FUNCTION_BLOCK PalletizerRemoteCtrl
VAR_INPUT
	bExecute : BOOL;
END_VAR
VAR_IN_OUT
	fbPalletizer : Palletizer;
END_VAR
VAR_OUTPUT
END_VAR
VAR
	
	udiStep : UDINT;
	messageIndex : UINT;
	remoteCtrlPayload : ST_MqttPayload;
	
	eActuatorType : E_ActuatorType;

END_VAR

(*

Description:
========================================================================	
	
	+	check if AdsConnector is connected
	+	if connected, subscribe to PalHmi topic
	+	check for incoming messages
	+	if message available, check message type 
	+	possible message types are:
	
			+	mode manual
			
				+	actuator type
				
					+	Belt
						+	forware
						+	backward
						
					+	Chain
						+	forward
						+	backward	
						
					+	BeltConveyor
						+	forward
						+	backward
						+	velocity
						
					+	RollerConveyor
						+	forward
						+	backward
						+	velocity	
						
					+	Turn
						+	forward
						+	backward
						
					+	Clamper
						+	clamp
						+	unclamp
	
					+	Pusher
						+	push forward
						+	push backward
						
					+	Plate
						+	open plate
						+	close plate
						
					+	Elevator
						+	up
						+	down
						+	to limit
						
			+	mode automatic
				
				+	start
				+	stop
			
			+	mode system
			
				+	home
				+	reset
				
			
=========================================================================

*)



IF 	ADS.fbAdsConnector.isConnected
	AND bExecute
THEN

	udiStep := 10;
ELSE
	udiStep := 0;
END_IF

CASE udiStep OF

	10:
		IF ADS.fbMqttClient.subscribe('PalHmi',THIS)
		THEN
			udiStep := 20;
		END_IF
		
	20:
		messageIndex := ADS.fbMqttClient.isNewMessage('PalHmi');
		IF messageIndex > 0
		THEN
		
			evaluateMode(Ads.fbMqttClient.getNewMessage(messageIndex));
			
		END_IF
			
		
END_CASE

METHOD PRIVATE evaluateActuator : BOOL
VAR_INPUT
	remoteCtrlPayload : ST_MqttPayload;
END_VAR
VAR
	eCmd : E_ActuatorCmdType;
	eActuator : E_ActuatorType;
END_VAR
eActuator := BYTE_TO_UINT(remoteCtrlPayload.data[2]);
eCmd := BYTE_TO_UINT(remoteCtrlPayload.data[3]);

CASE eActuator OF

	ePALLETIZER_BELT:
		
		fbPalletizer.fbBeltConveyor.cmd := eCmd;
		
	ePALLETIZER_CHAIN:
	
		fbPalletizer.fbPalletizerChain.cmd := eCmd;
		
	eBELT_CONVEYOR:
		
		fbPalletizer.fbBeltConveyor.cmd := eCmd;
		
	eROLLER_CONVEYOR:
		
		fbPalletizer.fbRollerConveyor.cmd := eCmd;
		
	eTURN_CYLINDER:
		
		fbPalletizer.fbTurnCylinder.cmd := eCmd;
	
	eCLAMPER_CYLINDER:
		
		fbPalletizer.fbClamperCylinder.cmd := eCmd;
	
	ePUSHER_CYLINDER:
		
		fbPalletizer.fbPusherCylinder.cmd := eCmd;
	
	ePLATE_CYLINDER:
		
		fbPalletizer.fbPlateCylinder.cmd := eCmd;
		
	eELEVATOR:
	
		fbPalletizer.fbElevator.cmd := eCmd;
	
END_CASE
END_METHOD

METHOD PRIVATE evaluateMode : BOOL
VAR_INPUT
	remoteCtrlPayload : ST_MqttPayload;
END_VAR
VAR	
	eCmd : E_ActuatorCmdType;
	eMode : E_ModeType;
END_VAR
(*
	data : ARRAY[1..32] OF Byte;
	
	data[1] -> mode type
	data[2] -> actutator type
	data[3] -> cmd
*)

eMode := BYTE_TO_UINT(remoteCtrlPayload.data[1]);
eCmd := BYTE_TO_UINT(remoteCtrlPayload.data[3]);

CASE eMode OF

	eAUTOMATIC_MODE_TYPE,
	eSYSTEM_MODE_TYPE:
		fbPalletizer.cmd := eCmd;
	eMANUAL_MODE_TYPE:
		evaluateActuator(remoteCtrlPayload);
	
END_CASE
END_METHOD

END_FUNCTION_BLOCK

(* stored: Version 1.1.0.1, ProductVersion 3.1.4024.2
   POU PalletizerRemoteCtrl: Id {d0ee27fa-3663-47e0-b662-636212931937}, SpecialFunc None
   Method evaluateActuator: Id {918ba018-8d14-4134-9588-6e91f6d5c994}
   Method evaluateMode: Id {6ea5a6ab-3f7d-4c18-a37b-cf49a7477800} *)
